PROGRAM PRG_TravelToSchool
VAR
END_VAR

END_PROGRAM

(* stored: Version 1.1.0.1, ProductVersion 3.1.4024.15
   POU PRG_TravelToSchool: Id {509033ce-6c15-471f-96e8-ab489b83a6fb}, SpecialFunc None *)
